// TIA Portal V17 export
// export: Created 2024-01-30T08:49:17.3499627Z, ExportSetting WithDefaults, DisplayName Totally Integrated Automation Portal, DisplayVersion V17 Update 6, DisplayName TIA Portal Openness, DisplayVersion V17 Update 6, DisplayName TIA Portal Version Control Interface, DisplayVersion V17, DisplayName STEP 7 Professional, DisplayVersion V17 Update 6, DisplayName STEP 7 Safety, DisplayVersion V17 Update 6, DisplayName WinCC Advanced, DisplayVersion V17 Update 6
TYPE "UDT_FESTO_CMMT_OUT"
// stored: IsFailsafeCompliant false
   STRUCT
      AxisEnabled : Bool;
      AxisPosOk : Bool;
      AxisSpFixed : Bool;
      AxisAckSetpoint : Bool;
      ClampTorqueReached : Bool;
      AxisRef : Bool;
      AxisWarn : Bool;
      AxisError : Bool;
      Lockout : Bool;
      ActVelocity : Real;
      ActPosition : DInt;
      ActMode : Int;
      EPosZSW1 : Word;
      EPosZSW2 : Word;
      ActWarn : Word;
      ActFault : Word;
      Error : Bool;
      Status : Word;
      DiagID : Word;
   END_STRUCT;
END_TYPE
